// TIA Portal V20 export
TYPE "LKinCtrl_bufferElement"
   STRUCT
      pathDataName : String["LKINCTRL_LENGTH_OF_PATHDATA_NAME"];
      pathDataIdentifier : USInt;
      setNumber : DInt;
      MotionType : Int := -1;
      MotionFBNo : Int;
      coordinateSystem : Int;
      transitionParameter : LReal;
      bufferMode : Int;
      measurementCmd : USInt;
      position : Array[1..6] of LReal;
   END_STRUCT;
END_TYPE
